SUBAPPLICATION Uebung_140_AX (* Übung zu SYS_ONTIME (Betriebsstundenzähler) *)
  (* Standard: 61499-2; Description: Copyright (c) 2026 Meisterschulen am Ostbahnhof This program and the accompanying materials are made available under the terms of the Eclipse Public License 2.0 which is available at https://www.eclipse.org/legal/epl-2.0/ SPDX-License-Identifier: EPL-2.0 *)
  (* Version 1.0, 2026-09-10, Franz Höpfinger, Meisterschulen am Ostbahnhof, initial API and implementation and/or initial documentation *)
  PACKAGE Uebungen;
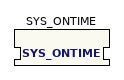
  FBS
    SYS_ONTIME : logiBUS::signalprocessing::measurement::SYS_ONTIME;
  END_FBS
END_SUBAPPLICATION
